// GVLs/HgGVL_Errors
// Contains common shared errors used in the mercury framework.
{attribute 'qualified_only'}
VAR_GLOBAL CONSTANT
	NO_ERROR 					: HgT_Error := HgF_CreateError(FALSE,HgE_ErrorCodes.ERR_NO_ERROR, 'No Error.', 0);
	TYPE_MISMATCH 				: HgT_Error := HgF_CreateError(TRUE, HgE_ErrorCodes.ERR_TYPE_MISMATCH, 'Type mismatch.', 0);
	SIZE_MISMATCH				: HgT_Error := HgF_CreateError(TRUE, HgE_ErrorCodes.ERR_SIZE_MISMATCH, 'Size mismatch.', 0);
	OUT_OF_BOUNDS				: HgT_Error := HgF_CreateError(TRUE, HgE_ErrorCodes.ERR_OUT_OF_BOUNDS, 'Value is outside the valid range.', 0);
	INVALID_INTERFACE  			: HgT_Error := HgF_CreateError(TRUE, HgE_ErrorCodes.ERR_INVALID_INTERFACE, 'Invalid or unknown interface.', 0);
	INVALID_REFERENCE  			: HgT_Error := HgF_CreateError(TRUE, HgE_ErrorCodes.ERR_INVALID_REFERENCE, 'Dereferencing an IEC reference in IecVarAccess failed due to an invalid destination address, e.g., NULL.', 0);
	INVALID_POINTER  			: HgT_Error := HgF_CreateError(TRUE, HgE_ErrorCodes.ERR_INVALID_POINTER, 'Invalid pointer.', 0);
	INVALID_CONVERSION  		: HgT_Error := HgF_CreateError(TRUE, HgE_ErrorCodes.ERR_INVALID_CONVERSION, 'Invalid data conversion.', 0);
	INVALID_COMPARISON  		: HgT_Error := HgF_CreateError(TRUE, HgE_ErrorCodes.ERR_INVALID_COMPARISON, 'Invalid comparison.', 0);
	INVALID_INPUT 				: HgT_Error := HgF_CreateError(TRUE, HgE_ErrorCodes.ERR_INVALID_INPUT, 'Invalid or unexpected input provided.', 0);
	MEMORY_ALLOCATION_FAILED 	: HgT_Error := HgF_CreateError(TRUE, HgE_ErrorCodes.ERR_MEMORY_ALLOCATION_FAILED, 'Memory allocation failed.', 0);
	INSUFFICIENT_MEMORY			: HgT_Error := HgF_CreateError(TRUE, HgE_ErrorCodes.ERR_INSUFFICIENT_MEMORY, 'Insufficient memory to carry out the request.', 0);
	OPERATION_FAILED			: HgT_Error := HgF_CreateError(TRUE, HgE_ErrorCodes.ERR_OPERATION_FAILED, 'Operation failed.', 0);
	INVALID_OPERATION			: HgT_Error := HgF_CreateError(TRUE, HgE_ErrorCodes.ERR_INVALID_OPERATION, 'Invalid Operation.', 0);
END_VAR

// PARAMs/HgPARAM_Constants
{attribute 'qualified_only'}
VAR_GLOBAL CONSTANT
	STR_SIZE : HgT_Size := 80; // Size of general string.
	SSTR_SIZE : HgT_Size := 40; // Size of short string.
	LSTR_SIZE : HgT_Size := 255; // Size of long string.
	INFO_SCAN_SIZE : HgT_Size := 15_000; // How many bytes to scan when looking for information. e.g. it's used by HgFB_Object to find the size of a child object in static memory.
END_VAR

// Version/Global_Version
{attribute 'TcGenerated'}
{attribute 'no-analysis'}
{attribute 'linkalways'}
// This function has been automatically generated from the project information.
VAR_GLOBAL CONSTANT
	{attribute 'const_non_replaced'}
	stLibVersion_Hg_Core : ST_LibVersion := (iMajor := 0, iMinor := 0, iBuild := 0, iRevision := 17, nFlags := 0, sVersion := '0.0.0.17');
END_VAR

// ITFs/HgI_Cloneable
INTERFACE HgI_Cloneable EXTENDS HgI_Object

// Creates a clone of the current object in dynamic memory.
METHOD Clone : HgI_Object
VAR_OUTPUT
	e : HgT_Error;
END_VAR
END_METHOD

END_INTERFACE

// ITFs/HgI_Object
// Generic interface that defines the basic properties and methods of an object in the mercury framework.
INTERFACE HgI_Object EXTENDS HgI_Queryable

// Pointer to the object in memory.
PROPERTY Address : HgT_Ptr
GET
END_GET
END_PROPERTY

// Gets the instance name of the object.
// NOTE: This only works of the object is in static memory.
METHOD GetInstanceName : HgT_LStr
VAR_OUTPUT
	e : HgT_Error;
END_VAR
END_METHOD

// Gets the instance path of the object.
// NOTE: This only works of the object is in static memory.
METHOD GetInstancePath : HgT_LStr
VAR_OUTPUT
	e : HgT_Error;
END_VAR
END_METHOD

// Returns a string representation of the object.
METHOD GetString : HgT_LStr
VAR_OUTPUT
	e : HgT_Error;
END_VAR
END_METHOD

// Gets the type name of the object as a string.
METHOD GetTypeName : HgT_Str
VAR_OUTPUT
	e : HgT_Error;
END_VAR
END_METHOD

// Checks if the current object is the same as (reference-wise) object as the input object.
METHOD Is : BOOL
VAR_INPUT
	ipObject : HgI_Object;
END_VAR
END_METHOD

// Memory area that the object is allocated in.
PROPERTY MemoryArea : HgT_MemArea
GET
END_GET
END_PROPERTY

//  Size of the object in bytes.
PROPERTY Size : HgT_Size
GET
END_GET
END_PROPERTY

END_INTERFACE

// ITFs/HgI_Queryable
// Root interface of all objects in the mercury framework. 
// Inherits __SYSTEM.IQueryInterface which is used to query an object interface/pointer for one of its interfaces.
INTERFACE HgI_Queryable EXTENDS __SYSTEM.IQueryInterface

END_INTERFACE

// ITFs/HgI_Configurable
// Base interface for a configurable system.
INTERFACE HgI_Configurable EXTENDS HgI_Object

END_INTERFACE

// ITFs/HgI_Configurator
// Base interface for a system configurator.
INTERFACE HgI_Configurator EXTENDS HgI_Object

END_INTERFACE

// ITFs/HgI_Controller
// Base interface for a controller.
INTERFACE HgI_Controller EXTENDS HgI_Object

END_INTERFACE

// ITFs/HgI_CopyableFrom
INTERFACE HgI_CopyableFrom EXTENDS HgI_Object

// Copies data to the current object from another object. Returns reference to self for method chaining.
METHOD CopyFrom : HgI_CopyableFrom
VAR_INPUT
	ipObject : HgI_Object; // Object to copy data from.
END_VAR
VAR_OUTPUT
	e : HgT_Error;
END_VAR
END_METHOD

END_INTERFACE

// ITFs/HgI_CopyableTo
INTERFACE HgI_CopyableTo EXTENDS HgI_Object

// Copies data from the current object to another object. Returns reference to self for method chaining.
METHOD CopyTo : HgI_CopyableTo
VAR_INPUT
	ipObject : HgI_Object; // Object to copy data to.
END_VAR
VAR_OUTPUT
	e : HgT_Error;
END_VAR
END_METHOD

END_INTERFACE

// ITFs/HgI_Error
// General interface for error classes in the mercury framework.
INTERFACE HgI_Error EXTENDS HgI_Queryable

// Error code specific to the particular error.
PROPERTY Code : HgT_ErrCode
GET
END_GET
END_PROPERTY

// Textual information describing the error.
PROPERTY Source : HgT_LStr
GET
END_GET
END_PROPERTY

// Indicates if an error has occurred | TRUE = error, FALSE = no error.
PROPERTY Status : BOOL
GET
END_GET
END_PROPERTY

END_INTERFACE

// ITFs/HgI_ErrorBuilder
// Interface for an error builder.
INTERFACE HgI_ErrorBuilder EXTENDS HgI_Object

// Appends the instance path of the caller to the source in the format <Caller::{caller instance path}>.
// NOTE: If the caller's interface is invalid; i.e. ipObject = 0, it will be ignored. 
METHOD AppendCallerToSource : HgI_ErrorBuilder
VAR_INPUT
	ipCaller : HgI_Object;
END_VAR
END_METHOD

// Appends a string to the error source.
METHOD AppendToSource : HgI_ErrorBuilder
VAR_INPUT
	Value : HgT_LStr;
END_VAR
END_METHOD

// Error code specific to the particular error.
PROPERTY Code : HgT_ErrCode
GET
END_GET
SET
END_SET
END_PROPERTY

// Returns the built error.
METHOD GetError : HgFB_Error
VAR_INPUT
END_VAR
END_METHOD

// Prepends a string to the error source.
METHOD PrependToSource : HgI_ErrorBuilder
VAR_INPUT
	Value : HgT_LStr;
END_VAR
END_METHOD

// Resets the built error.
METHOD Reset : HgI_ErrorBuilder
VAR_INPUT
END_VAR
END_METHOD

// Sets the error code of the error.
METHOD SetCode : HgI_ErrorBuilder
VAR_INPUT
	Code : HgT_ErrCode;
END_VAR
END_METHOD

// Sets the error in the error builder.
METHOD SetError : HgI_ErrorBuilder
VAR_INPUT
	Error : HgT_Error;
END_VAR
END_METHOD

// Sets the error source of the error.
METHOD SetSource : HgI_ErrorBuilder
VAR_INPUT
	Source : HgT_LStr;
END_VAR
END_METHOD

// Sets the status of the error
METHOD SetStatus : HgI_ErrorBuilder
VAR_INPUT
	bStatus : BOOL;
END_VAR
END_METHOD

// Textual information describing the error.
PROPERTY Source : HgT_LStr
GET
END_GET
SET
END_SET
END_PROPERTY

// Indicates if an error has occurred | TRUE = error, FALSE = no error.
PROPERTY Status : BOOL
GET
END_GET
SET
END_SET
END_PROPERTY

END_INTERFACE

// POUs/Function Blocks/HgFB_Error
// HgFB_Error is the base function block used for error handling and reporting within the mercury framework.
{attribute 'enable_dynamic_creation'}
{attribute 'no_explicit_call' := 'direct call for this function block is not allowed'}
FUNCTION_BLOCK HgFB_Error IMPLEMENTS HgI_Error
VAR
	_Status : BOOL;
	_Code : HgT_ErrCode;
	_Source : HgT_LStr;
END_VAR

// Error code specific to the particular error.
PROPERTY Code : HgT_ErrCode
GET
Code := THIS^._Code;
END_GET
END_PROPERTY

// Textual information describing the error.
PROPERTY Source : HgT_LStr
GET
Source := THIS^._Source;
END_GET
END_PROPERTY

// Indicates if an error has occurred | TRUE = error, FALSE = no error.
PROPERTY Status : BOOL
GET
Status := THIS^._Status;
END_GET
END_PROPERTY

END_FUNCTION_BLOCK

// ITFs/HgI_Status
// Base interface for a system status information.
INTERFACE HgI_Status EXTENDS HgI_Object

END_INTERFACE

// ITFs/HgI_StatusProvider
// Base interface for a system that can provide status.
INTERFACE HgI_StatusProvider EXTENDS HgI_Object

END_INTERFACE

// POUs/Function Blocks/HgFB_CycleChanged
// Function block that can be used to indicate if a the current task cycle it is instantated at has changed.
{attribute 'enable_dynamic_creation'}
{attribute 'reflection'}
{attribute 'no_explicit_call' := 'direct call for this function block is not allowed'} 
FUNCTION_BLOCK FINAL HgFB_CycleChanged EXTENDS HgFB_Object
VAR
	_nCycleLastCalled : UDINT := 4294967295; // The last cycle checked for change-in-plc-cycle.
	_nTaskIndex : DINT := HgF_GetPlcTaskInformation().TaskIndex; // The task index the function block was instantiated on.
END_VAR

// A string that represents the type of the object if the object is created dynamically.
// Function blocks intended for dynamic use must override this property.
PROPERTY PROTECTED DynamicTypeName : HgT_Str
GET
DynamicTypeName := 'HgFB_CycleChanged';
END_GET
END_PROPERTY

// Flag to indicate if cycle the cycle the function block was instantiated at has changed | TRUE = Cycle has changed.
PROPERTY _ : BOOL
GET
VAR
	nTmp : UDINT;
END_VAR
nTmp := THIS^.GetCurrentCycle();

_ := THIS^.CycleLastChecked <> nTmp;

THIS^._nCycleLastCalled := nTmp;
END_GET
END_PROPERTY

// The last cycle checked for change-in-plc-cycle.
PROPERTY CycleLastChecked : UDINT
GET
CycleLastChecked := THIS^._nCycleLastCalled;
END_GET
END_PROPERTY

// Indicates whether this is the first cycle of the task the function block was instatiated at | TRUE = first cycle.
PROPERTY FirstCycle : BOOL
GET
 FirstCycle := TwinCAT_SystemInfoVarList._TaskInfo[THIS^._nTaskIndex].FirstCycle;
END_GET
END_PROPERTY

// The current cycle of the task the function block was instatiated on.
METHOD GetCurrentCycle : UDINT
VAR_INPUT
END_VAR
GetCurrentCycle := TwinCAT_SystemInfoVarList._TaskInfo[THIS^._nTaskIndex].CycleCount;
END_METHOD

// Returns a string representation of the object.
METHOD GetString : HgT_LStr
VAR_OUTPUT
	e : HgT_Error;
END_VAR
GetString := TO_STRING(THIS^._);
END_METHOD

// Size of the object in bytes.
PROPERTY Size : HgT_Size
GET
Size := SIZEOF(THIS^);
END_GET
END_PROPERTY

// The task index the function block is instatiated on.
PROPERTY TaskIndex : DINT
GET
TaskIndex := THIS^._nTaskIndex;
END_GET
END_PROPERTY

END_FUNCTION_BLOCK

// POUs/Function Blocks/HgFB_Object
// Base function block of all mercury function blocks in the mercury framework.
{attribute 'enable_dynamic_creation'}
{attribute 'reflection'}
{attribute 'no_assign'}
{attribute 'no_explicit_call' := 'direct call for this function block is not allowed'} 
FUNCTION_BLOCK HgFB_Object IMPLEMENTS HgI_Object
VAR
END_VAR

// A string that represents the type of the object if the object is created dynamically.
// Function blocks intended for dynamic use must override this property.
PROPERTY PROTECTED DynamicTypeName : HgT_Str
GET
DynamicTypeName := 'HgFB_Object';
END_GET
END_PROPERTY

// Private local variable that acts as a flag to indicate that the size of the object may need to be recomputed.
PROPERTY PRIVATE RecomputeSize : REFERENCE TO BOOL
GET
VAR_INST
	bRecomputeSize : BOOL;
END_VAR
RecomputeSize REF= bRecomputeSize;
END_GET
END_PROPERTY

// Pointer to the object in memory.
PROPERTY FINAL Address : HgT_Ptr
GET
Address := THIS;
END_GET
END_PROPERTY

{attribute 'hide'}
METHOD FB_init : BOOL
VAR_INPUT
	bInitRetains : BOOL; // if TRUE, the retain variables are initialized (warm start / cold start)
	bInCopyCode : BOOL;  // if TRUE, the instance afterwards gets moved into the copy code (online change)
END_VAR
// Raise the recompute size flag whenever an online change is made.
// Please don't remove the 'IF' block because you think it should be 'THIS^.RecomputeSize := bInCopyCode;'
// This is done on purpose to latch the flag. Only the size property should reset it.
IF bInCopyCode THEN THIS^.RecomputeSize := bInCopyCode; END_IF
END_METHOD

{attribute 'hide'}
METHOD FB_reinit : BOOL
VAR_INPUT
END_VAR
END_METHOD

// Gets the instance name of the object.
// NOTE: This only works of the object is in static memory.
METHOD FINAL GetInstanceName : HgT_LStr
VAR_OUTPUT
	e : HgT_Error;
END_VAR
CASE THIS^.MemoryArea OF
	HgT_MemArea.Static: 
		GetInstanceName := HgF_GetVariableNameByAddress(THIS, THIS^.Size, e => e);
	HgT_MemArea.Dynamic:
		GetInstanceName := '<Dynamic>';
	HgT_MemArea.CNC:
		GetInstanceName := '<Unsupported>';
ELSE
	GetInstanceName := '<Unknown>';
	e := HgF_CreateError(TRUE, HgE_ErrorCodes.ERR_OPERATION_FAILED, 'Cannot identify the memory area of the object.', 0);
	END_CASE
END_METHOD

// Gets the instance path of an object.
// NOTE: This only works of the object is in static memory.
METHOD FINAL GetInstancePath : HgT_LStr
VAR_OUTPUT
	e : HgT_Error;
END_VAR
CASE THIS^.MemoryArea OF
	HgT_MemArea.Static: 
		GetInstancePath := HgF_GetVariablePathByAddress(THIS, THIS^.Size, e => e);
	HgT_MemArea.Dynamic:
		GetInstancePath := '<Dynamic>';
	HgT_MemArea.CNC:
		GetInstancePath := '<Unsupported>';
ELSE
	GetInstancePath := '<Unknown>';
	e := HgF_CreateError(TRUE, HgE_ErrorCodes.ERR_OPERATION_FAILED, 'Cannot identify the memory area of the object.', 0);
	END_CASE
END_METHOD

// Returns a string representation of the object.
{attribute 'TcRpcEnable'}
METHOD GetString : HgT_LStr
VAR_OUTPUT
	e : HgT_Error;
END_VAR
GetString := THIS^.GetTypeName(e => e);

IF e.Status THEN RETURN; END_IF

GetString := Tc2_Standard.CONCAT(GetString, CONCAT(' at ', TO_STRING(THIS)));
END_METHOD

// Gets the type name of the object as a string.
METHOD FINAL GetTypeName : HgT_Str
VAR_OUTPUT
	e : HgT_Error;
END_VAR
CASE THIS^.MemoryArea OF
	HgT_MemArea.Static: 
		GetTypeName := HgF_GetTypeNameByAddress(THIS, THIS^.Size, e => e);
	HgT_MemArea.Dynamic:
		GetTypeName := THIS^.DynamicTypeName;
	HgT_MemArea.CNC:
		GetTypeName := '<Unsupported>';
ELSE
	GetTypeName := '<Unknown>';
	END_CASE
END_METHOD

// Checks if the current object is the same as (reference-wise) object as the input object.
METHOD FINAL Is : BOOL
VAR_INPUT
	ipObject : HgI_Object;
END_VAR
Is := SEL(ipObject <> 0, FALSE, ipObject.Address = THIS);
END_METHOD

// Memory area that the object is allocated in.
PROPERTY FINAL MemoryArea : HgT_MemArea
GET
MemoryArea := Tc2_System.F_CheckMemoryArea(THIS, 1);
END_GET
END_PROPERTY

// Size of the object in bytes.
PROPERTY Size : HgT_Size
GET
VAR_INST
	_Size : HgT_Size;
END_VAR
IF _Size > 0 AND NOT(THIS^.RecomputeSize) THEN Size := _Size; RETURN; END_IF

// Set the recompute flag to false.
THIS^.RecomputeSize := FALSE;

CASE THIS^.MemoryArea OF
// Attempt to get size of object.
	HgT_MemArea.Static:
	// If object is in static memory try and look for it using the TcCOM object server and get it's size.
		FOR _Size := SIZEOF(THIS^) TO HgPARAM_Constants.INFO_SCAN_SIZE DO
			IF HgF_GetTypeNameByAddress(THIS, _Size) <> '' THEN RETURN; END_IF
			END_FOR
	END_CASE
	
// In any other case just return the base object size.
_Size := SIZEOF(THIS^);
END_GET
END_PROPERTY

END_FUNCTION_BLOCK

// POUs/Functions/HgF_GetVariableNameByAddress
// Returns the name of a variable as a string using its pointer and size.
// Variables allocated in dynamic memory are not supported.
FUNCTION HgF_GetVariableNameByAddress : HgT_LStr
VAR_INPUT
	Address : HgT_Ptr; // Pointer to variable.
	Size : HgT_Size; // Size of variable in bytes.
END_VAR
VAR_OUTPUT
	e : HgT_Error;
END_VAR
VAR
	_pCursor : POINTER TO BYTE;
	_pVariableName : POINTER TO HgT_LStr;
END_VAR

HgF_GetVariableNameByAddress := HgF_GetVariablePathByAddress(Address, Size, e => e);

IF e.Status OR_ELSE HgF_GetVariableNameByAddress = '' THEN RETURN; END_IF

_pCursor := ADR(HgF_GetVariableNameByAddress);

REPEAT
	IF _pCursor^ = 46 THEN _pVariableName := _pCursor + 1; END_IF
	_pCursor := _pCursor + 1;
UNTIL
	_pCursor^ = 0
	END_REPEAT

HgF_GetVariableNameByAddress := SEL(_pVariableName = 0, _pVariableName^, HgF_GetVariableNameByAddress);

END_FUNCTION

// POUs/Functions/HgF_GetVariablePathByAddress
// Returns the path of a variable as a string using its pointer and size.
// Variables allocated in dynamic memory are not supported.
{warning disable C0394}
FUNCTION HgF_GetVariablePathByAddress : HgT_LStr
VAR_INPUT
	Address : HgT_Ptr; // Pointer to variable.
	Size : HgT_Size; // Size of variable in bytes.
END_VAR
VAR_OUTPUT
	e : HgT_Error;
END_VAR
VAR
	_nTmp : UDINT := SIZEOF(HgF_GetVariablePathByAddress);
	_ipComInterface : ITcIecApplicationInfo := HgF_TcComIecApplicationInfo().GetInterface(e => e);;
	_Result : HRESULT;
END_VAR

IF _ipComInterface <> 0 THEN
	_Result := _ipComInterface.GetSymbolNameByAddress(TO_UDINT(Size), Address, _nTmp, ADR(HgF_GetVariablePathByAddress));
	e := SEL(
		Tc3_Module.SUCCEEDED(_Result),
		HgF_CreateError(TRUE, _Result, 'Failed to get variable path. Check error code against "Tc3_Module/Error Codes" section on infosys.', 0),
		HgGVL_Errors.NO_ERROR);
	END_IF

END_FUNCTION

// POUs/Functions/HgF_CreateError
// Function for creating an error function block.
// If ipObject object is not 0 the instance path will be appended to the error message.
FUNCTION HgF_CreateError : HgFB_Error
VAR_INPUT
	bStatus : BOOL; // Indicates if an error has occurred | TRUE = error, FALSE = no error.
	Code : HgT_ErrCode; // Error code specific to the particular error.
	Source : HgT_LStr; // Textual information describing the error.
	ipCaller : HgI_Object; // Object that created the error, set to 0 if you don't want append caller to error message.
END_VAR
VAR
	_fbError : HgFB_MutableError;
END_VAR

_fbError.Status := bStatus;
_fbError.Code := Code;
_fbError.Source := Source;

HgF_CreateError := _fbError.AppendCaller(ipCaller);

END_FUNCTION

// POUs/Function Blocks/HgFB_MutableError
// Base function block for mutable errors used for error handling and reporting within the mercury framework.
{attribute 'enable_dynamic_creation'}
{attribute 'no_explicit_call' := 'direct call for this function block is not allowed'}
FUNCTION_BLOCK HgFB_MutableError EXTENDS HgFB_Error IMPLEMENTS HgI_Error
VAR
END_VAR

METHOD FINAL AppendCaller : REFERENCE TO HgFB_MutableError
VAR_INPUT
	ipCaller : HgI_Object;
END_VAR
AppendCaller REF= THIS^;
IF ipCaller = 0 THEN RETURN; END_IF

THIS^._Source := CONCAT(THIS^._Source, CONCAT(' <Caller::', CONCAT(ipCaller.GetInstancePath(),'>')));
END_METHOD

// Error code specific to the particular error.
PROPERTY FINAL Code : HgT_ErrCode
SET
THIS^._Code := Code;
END_SET
END_PROPERTY

// Textual information describing the error.
PROPERTY FINAL Source : HgT_LStr
SET
THIS^._Source := Source;
END_SET
END_PROPERTY

// Indicates if an error has occurred | TRUE = error, FALSE = no error.
PROPERTY FINAL Status : BOOL
SET
THIS^._Status := Status;
END_SET
END_PROPERTY

END_FUNCTION_BLOCK

// POUs/Functions/HgF_TcComIecApplicationInfo
// Function that acts as a singleton for HgFB_TcComIecApplicationInfo, a function block that that manages the ITcIecApplicationInfo TcCOM Interface used by Hg_Core.
FUNCTION HgF_TcComIecApplicationInfo : REFERENCE TO HgFB_TcComIecApplicationInfo
VAR_STAT
	_fbTcComIecApplicationInfo : HgFB_TcComIecApplicationInfo;
END_VAR

HgF_TcComIecApplicationInfo REF= _fbTcComIecApplicationInfo;

END_FUNCTION

// POUs/Function Blocks/HgFB_TcComIecApplicationInfo
// Function block that manages the ITcIecApplicationInfo TcCOM Interface used by Hg_Core.
{attribute 'enable_dynamic_creation'}
{attribute 'no_assign'}
{attribute 'no_explicit_call' := 'direct call for this function block is not allowed'} 
FUNCTION_BLOCK FINAL HgFB_TcComIecApplicationInfo IMPLEMENTS HgI_Queryable
VAR
	_ipIecApplicationInformation : ITcIecApplicationInfo;
	_hIecApplicationInformation : HRESULT := Tc3_Module.GVL.E_FAIL;
END_VAR

{attribute 'hide'}
METHOD FB_exit : BOOL
VAR_INPUT
	bInCopyCode : BOOL; // if TRUE, the exit method is called for exiting an instance that is copied afterwards (online change).
END_VAR
// no online change
IF bInCopyCode THEN RETURN; END_IF

// Safe release of ITcIecApplicationInfo.
Tc3_Module.FW_SafeRelease(ADR(THIS^._ipIecApplicationInformation));
THIS^._hIecApplicationInformation := Tc3_Module.GVL.E_FAIL;
END_METHOD

{attribute 'hide'}
{attribute 'no_explicit_call' := 'direct call for this method is not allowed'}
METHOD FB_init : BOOL
VAR_INPUT
	bInitRetains : BOOL; // if TRUE, the retain variables are initialized (warm start / cold start)
	bInCopyCode : BOOL;  // if TRUE, the instance afterwards gets moved into the copy code (online change)
END_VAR
// No online change.
IF bInCopyCode THEN RETURN; END_IF

// Get instance of ITcIecApplicationInfo.
THIS^._hIecApplicationInformation := Tc3_Module.FW_ObjMgr_GetObjectInstance(
	TwinCAT_SystemInfoVarList._AppInfo.ObjId, 
	TC_GLOBAL_IID_LIST.IID_ITcIecApplicationInfo, 
	ADR(THIS^._ipIecApplicationInformation)
);
END_METHOD

METHOD GetInterface : ITcIecApplicationInfo
VAR_OUTPUT
	e : HgT_Error;
END_VAR
// If instance of ITcIecApplicationInfo failed to be obtained on 
// FB_init or FB_exit was explicitly called try to get it gain.


IF Tc3_Module.FAILED(THIS^._hIecApplicationInformation) THEN
	THIS^._hIecApplicationInformation := Tc3_Module.FW_ObjMgr_GetObjectInstance(
		TwinCAT_SystemInfoVarList._AppInfo.ObjId, 
		TC_GLOBAL_IID_LIST.IID_ITcIecApplicationInfo, 
		ADR(THIS^._ipIecApplicationInformation)
	);
	END_IF

e := SEL(
	Tc3_Module.SUCCEEDED(THIS^._hIecApplicationInformation),
	HgF_CreateError(TRUE, THIS^._hIecApplicationInformation, 'No failed to get interface. Check error code against "Tc3_Module/Error Codes" section on infosys.', 0),
	HgGVL_Errors.NO_ERROR);

GetInterface := THIS^._ipIecApplicationInformation;
END_METHOD

END_FUNCTION_BLOCK

// POUs/Functions/HgF_GetTypeNameByAddress
// Returns the datatype of a variable as a string using its pointer and size.
// Variables allocated in dynamic memory are not supported.
FUNCTION HgF_GetTypeNameByAddress : HgT_Str
VAR_INPUT
	Address :HgT_Ptr; // Pointer to variable.
	Size : HgT_Size; // Size of variable in bytes.
END_VAR
VAR_OUTPUT
	e : HgT_Error;
END_VAR
VAR 
	_nTmp : UDINT := SIZEOF(HgF_GetTypeNameByAddress);
	_ipComInterface : ITcIecApplicationInfo := HgF_TcComIecApplicationInfo().GetInterface(e => e);;
	_Result : HRESULT;
END_VAR


	
IF _ipComInterface <> 0 THEN
	_Result := _ipComInterface.GetDatatypeNameByAddress(TO_UDINT(Size), Address, _nTmp, ADR(HgF_GetTypeNameByAddress));
	e := SEL(
		Tc3_Module.SUCCEEDED(_Result),
		HgF_CreateError(TRUE, _Result, 'Failed to get variable typename. Check error code against "Tc3_Module/Error Codes" section on infosys.', 0),
		HgGVL_Errors.NO_ERROR);
	END_IF

END_FUNCTION

// POUs/Functions/HgF_GetPlcTaskInformation
// Retrieves the current plc task's information.
FUNCTION HgF_GetPlcTaskInformation : REFERENCE TO HgT_PlcTaskInfo
VAR
	_fbGetCurrentTaskIndex : GETCURTASKINDEX;
	_PlcTaskSysInfo : PlcTaskSystemInfo;
END_VAR
VAR_STAT
	_PlcTaskInformation : HgT_PlcTaskInfo;
END_VAR

_fbGetCurrentTaskIndex();
_PlcTaskSysInfo := TwinCAT_SystemInfoVarList._TaskInfo[_fbGetCurrentTaskIndex.index];
_PlcTaskInformation.AdsPort 				:= _PlcTaskSysInfo.AdsPort;
_PlcTaskInformation.CycleCount 				:= _PlcTaskSysInfo.CycleCount;
_PlcTaskInformation.CycleTime 				:= TO_LTIME(_PlcTaskSysInfo.CycleTime*100);
_PlcTaskInformation.CycleTimeExceeded 		:= _PlcTaskSysInfo.CycleTimeExceeded;
_PlcTaskInformation.DcTaskTime 				:= _PlcTaskSysInfo.DcTaskTime;
_PlcTaskInformation.FirstCycle				:= _PlcTaskSysInfo.FirstCycle;
_PlcTaskInformation.InCallAfterOutputUpdate := _PlcTaskSysInfo.InCallAfterOutputUpdate;
_PlcTaskInformation.LastExecTime 			:= TO_LTIME(_PlcTaskSysInfo.LastExecTime*100);
_PlcTaskInformation.ObjId 					:= _PlcTaskSysInfo.ObjId;
_PlcTaskInformation.Priority 				:= _PlcTaskSysInfo.Priority;
_PlcTaskInformation.RTViolation 			:= _PlcTaskSysInfo.RTViolation;
_PlcTaskInformation.TaskName 				:= _PlcTaskSysInfo.TaskName;
_PlcTaskInformation.TaskIndex 				:= _fbGetCurrentTaskIndex.Index;

HgF_GetPlcTaskInformation REF= _PlcTaskInformation;

END_FUNCTION

// POUs/Function Blocks/HgFB_ErrorBuilder
// Function block for building an error.
{attribute 'enable_dynamic_creation'}
{attribute 'no_explicit_call' := 'direct call for this function block is not allowed'} 
FUNCTION_BLOCK FINAL HgFB_ErrorBuilder EXTENDS HgFB_Object IMPLEMENTS HgI_ErrorBuilder
VAR
	// Working error.
	_Error : HgFB_MutableError;
END_VAR

// Appends the instance path of the caller to the source in the format <Caller::{caller instance path}>.
// NOTE: If the caller's interface is invalid; i.e. ipObject = 0, it will be ignored. 
METHOD AppendCallerToSource : HgI_ErrorBuilder
VAR_INPUT
	ipCaller : HgI_Object;
END_VAR
AppendCallerToSource := THIS^;

THIS^._Error.AppendCaller(ipCaller);
END_METHOD

// Appends a string to the error source.
METHOD AppendToSource : HgI_ErrorBuilder
VAR_INPUT
	Value : HgT_LStr;
END_VAR
AppendToSource := THIS^;

THIS^._Error.Source := Tc2_Standard.CONCAT(THIS^._Error.Source, Value);
END_METHOD

// Error code specific to the particular error.
PROPERTY Code : HgT_ErrCode
GET
Code := THIS^._Error.Code;
END_GET
SET
THIS^._Error.Code := Code;
END_SET
END_PROPERTY

// A string that represents the type of the object if the object is created dynamically.
// Function blocks intended for dynamic use must override this property.
PROPERTY PROTECTED DynamicTypeName : HgT_Str
GET
DynamicTypeName := 'HgFB_ErrorBuilder';
END_GET
END_PROPERTY

// Returns the built error.
{attribute 'TcRpcEnable'}
METHOD GetError : HgFB_Error
VAR_INPUT
END_VAR
GetError := THIS^._Error;
END_METHOD

// Returns a string representation of the object.
{attribute 'TcRpcEnable'}
{warning disable C0394}
METHOD GetString : HgT_LStr
VAR_OUTPUT
	e : HgT_Error;
END_VAR
VAR
	fbJson : Tc3_JsonXml.FB_JsonSaxWriter;
	Result : HRESULT;
END_VAR
fbJson.StartObject();
fbJson.AddKey('Status');
fbJson.AddBool(THIS^._Error.Status);
fbJson.AddKey('Code');
fbJson.AddLint(THIS^._Error.Code);
fbJson.AddKey('Source');
GetString := THIS^._Error.Source;
fbJson.AddString(GetString);
fbJson.EndObject();
GetString := fbJson.GetDocument(hrErrorCode => Result);
e := SEL(
	Tc3_Module.SUCCEEDED(Result),
	HgF_CreateError(TRUE, Result, 'Failed to generate json. Check error code against "Tc3_Module/Error Codes" section on infosys.', 0),
	HgGVL_Errors.NO_ERROR);
END_METHOD

// Prepends a string to the error source.
METHOD PrependToSource : HgI_ErrorBuilder
VAR_INPUT
	Value : HgT_LStr;
END_VAR
PrependToSource := THIS^;

THIS^._Error.Source := Tc2_Standard.CONCAT(Value, THIS^._Error.Source);
END_METHOD

// Resets the built error.
METHOD Reset : HgI_ErrorBuilder
VAR_INPUT
END_VAR
Reset := THIS^;

THIS^._Error.Status := FALSE;
THIS^._Error.Code := 0;
THIS^._Error.Source := '';
END_METHOD

// Sets the error code of the error.
METHOD SetCode : HgI_ErrorBuilder
VAR_INPUT
	Code : HgT_ErrCode;
END_VAR
SetCode := THIS^;

THIS^._Error.Code := Code;
END_METHOD

// Sets the error in the error builder.
METHOD SetError : HgI_ErrorBuilder
VAR_INPUT
	Error : HgT_Error;
END_VAR
SetError := THIS^;

THIS^._Error.Status := Error.Status;
THIS^._Error.Code := Error.Code;
THIS^._Error.Source := Error.Source;
END_METHOD

// Sets the error source of the error.
METHOD SetSource : HgI_ErrorBuilder
VAR_INPUT
	Source : HgT_LStr;
END_VAR
SetSource := THIS^;

THIS^._Error.Source := Source;
END_METHOD

// Sets the status of the error
METHOD SetStatus : HgI_ErrorBuilder
VAR_INPUT
	bStatus : BOOL;
END_VAR
SetStatus := THIS^;

THIS^._Error.Status := bStatus;
END_METHOD

PROPERTY Size : HgT_Size
GET
Size := SIZEOF(THIS^);
END_GET
END_PROPERTY

// Textual information describing the error.
PROPERTY Source : HgT_LStr
GET
Source := THIS^._Error.Source;
END_GET
SET
THIS^._Error.Source := Source;
END_SET
END_PROPERTY

// Indicates if an error has occurred | TRUE = error, FALSE = no error.
PROPERTY Status : BOOL
GET
Status := THIS^._Error.Status;
END_GET
SET
THIS^._Error.Status := Status;
END_SET
END_PROPERTY

END_FUNCTION_BLOCK

// POUs/Function Blocks/HgFB_FirstCall
// Function block that can be used to indicate whether a section of code has been running for the first time.
{attribute 'enable_dynamic_creation'}
{attribute 'reflection'}
{attribute 'no_explicit_call' := 'direct call for this function block is not allowed'} 
FUNCTION_BLOCK FINAL HgFB_FirstCall EXTENDS HgFB_Object
VAR
	_CallFlag : BOOL := TRUE; 
END_VAR

// Flag to indicate if code section is running for the first time | TRUE = Called for the first time.
PROPERTY _ : BOOL
GET
_ := THIS^._CallFlag;

THIS^._CallFlag := FALSE;
END_GET
END_PROPERTY

// A string that represents the type of the object if the object is created dynamically.
// Function blocks intended for dynamic use must override this property.
PROPERTY PROTECTED DynamicTypeName : HgT_Str
GET
DynamicTypeName := 'HgFB_FirstCall';
END_GET
END_PROPERTY

// Returns a string representation of the object.
METHOD GetString : HgT_LStr
VAR_OUTPUT
	e : HgT_Error;
END_VAR
GetString := TO_STRING(THIS^._);
END_METHOD

// Resets the flag for first call.
METHOD Reset
VAR_INPUT
END_VAR
THIS^._CallFlag := TRUE;
END_METHOD

PROPERTY Size : HgT_Size
GET
Size := SIZEOF(THIS^);
END_GET
END_PROPERTY

END_FUNCTION_BLOCK

// POUs/Function Blocks/HgFB_FlagHasChanged
// Checks if the watched value has changed.
{attribute 'enable_dynamic_creation'}
{attribute 'no_explicit_call' := 'direct call for this function block is not allowed'} 
FUNCTION_BLOCK FINAL HgFB_FlagHasChanged EXTENDS HgFB_Object
VAR
	_bValue : BOOL; 
END_VAR

// A string that represents the type of the object if the object is created dynamically.
// Function blocks intended for dynamic use must override this property.
PROPERTY PROTECTED DynamicTypeName : HgT_Str
GET
DynamicTypeName := 'HgFB_FlagHasChanged';
END_GET
END_PROPERTY

// Size of the object in bytes.
PROPERTY Size : HgT_Size
GET
Size := SIZEOF(THIS^);
END_GET
END_PROPERTY

METHOD Watch : BOOL
VAR_INPUT
	Value : BOOL;
END_VAR
VAR_INST
	bFirstCall : BOOL := TRUE;
END_VAR
IF bFirstCall THEN bFirstCall := FALSE; Watch := TRUE; THIS^._bValue := Value; RETURN; END_IF

Watch := THIS^._bValue <> Value;
END_METHOD

END_FUNCTION_BLOCK

// POUs/Function Blocks/HgFB_FloatHasChanged
// Checks if the watched value has changed.
{attribute 'enable_dynamic_creation'}
{attribute 'no_explicit_call' := 'direct call for this function block is not allowed'} 
FUNCTION_BLOCK FINAL HgFB_FloatHasChanged EXTENDS HgFB_Object
VAR
	_fValue : LREAL; 
END_VAR

// A string that represents the type of the object if the object is created dynamically.
// Function blocks intended for dynamic use must override this property.
PROPERTY PROTECTED DynamicTypeName : HgT_Str
GET
DynamicTypeName := 'HgFB_FloatHasChanged';
END_GET
END_PROPERTY

// Size of the object in bytes.
PROPERTY Size : HgT_Size
GET
Size := SIZEOF(THIS^);
END_GET
END_PROPERTY

METHOD Watch : BOOL
VAR_INPUT
	fValue : LREAL;
END_VAR
VAR_INST
	bFirstCall : BOOL := TRUE;
END_VAR
IF bFirstCall THEN bFirstCall := FALSE; Watch := TRUE; THIS^._fValue := fValue; RETURN; END_IF

Watch := THIS^._fValue <> fValue;
END_METHOD

END_FUNCTION_BLOCK

// POUs/Function Blocks/HgFB_HasChanged
// Checks if the watched value has changed.
{attribute 'enable_dynamic_creation'}
{attribute 'reflection'}
{attribute 'no_explicit_call' := 'direct call for this function block is not allowed'} 
FUNCTION_BLOCK FINAL HgFB_HasChanged EXTENDS HgFB_Object
VAR
	_nHash 		: DWORD;
	_nSize		: DINT 					:= -1;
	_eTypeClass : __SYSTEM.TYPE_CLASS 	:= __SYSTEM.TYPE_CLASS.TYPE_NONE;
END_VAR

// A string that represents the type of the object if the object is created dynamically.
// Function blocks intended for dynamic use must override this property.
PROPERTY PROTECTED DynamicTypeName : HgT_Str
GET
DynamicTypeName := 'HgFB_HasChanged';
END_GET
END_PROPERTY

// Size of the object in bytes.
PROPERTY Size : HgT_Size
GET
Size := SIZEOF(THIS^);
END_GET
END_PROPERTY

METHOD Watch : BOOL
VAR_INPUT
	Value : ANY;
END_VAR
VAR
	nHash : DWORD;
END_VAR
nHash := HgF_SimpleHash(Value);

IF THIS^._nHash = nHash AND_THEN THIS^._nSize = Value.diSize AND_THEN THIS^._eTypeClass = Value.TypeClass THEN RETURN; END_IF 

THIS^._nHash 		:= nHash;
THIS^._nSize 		:= Value.diSize;
THIS^._eTypeClass 	:= Value.TypeClass;

Watch := TRUE;
END_METHOD

END_FUNCTION_BLOCK

// POUs/Functions/HgF_SimpleHash
// This function calculates a hashcode of a given value using the FNV-1a 32-bit hash algorithm. Source: http://www.isthe.com/chongo/tech/comp/fnv/
FUNCTION HgF_SimpleHash : DWORD
VAR_INPUT
	Data : ANY;
END_VAR
VAR
	i, nSize, nHash : DWORD;
END_VAR
VAR_STAT CONSTANT
	nPrime : DWORD := 16#1000193; // 32-bit FNV Prime
END_VAR

nHash := 16#811C9DC5; // 32-bit offset basis
CASE Data.TypeClass OF
	__SYSTEM.TYPE_CLASS.TYPE_STRING:
		nSize := Tc2_Utilities.LEN2(Data.pValue)- 1;
	__SYSTEM.TYPE_CLASS.TYPE_WSTRING:
		nSize := Tc2_Utilities.WLEN2(Data.pValue)*2-1;
ELSE
		nSize := TO_UDINT(Data.diSize) - 1;
END_CASE
FOR i := 0 TO nSize DO nHash :=(nHash XOR Data.pValue[i])*nPrime; END_FOR
HgF_SimpleHash := nHash;

END_FUNCTION

// POUs/Function Blocks/HgFB_IntHasChanged
// Checks if the watched value has changed.
{attribute 'enable_dynamic_creation'}
{attribute 'no_explicit_call' := 'direct call for this function block is not allowed'} 
FUNCTION_BLOCK FINAL HgFB_IntHasChanged EXTENDS HgFB_Object
VAR
	_nValue : LINT; 
END_VAR

// A string that represents the type of the object if the object is created dynamically.
// Function blocks intended for dynamic use must override this property.
PROPERTY PROTECTED DynamicTypeName : HgT_Str
GET
DynamicTypeName := 'HgFB_IntHasChanged';
END_GET
END_PROPERTY

// Size of the object in bytes.
PROPERTY Size : HgT_Size
GET
Size := SIZEOF(THIS^);
END_GET
END_PROPERTY

METHOD Watch : BOOL
VAR_INPUT
	nValue : LINT;
END_VAR
VAR_INST
	bFirstCall : BOOL := TRUE;
END_VAR
IF bFirstCall THEN bFirstCall := FALSE; Watch := TRUE; THIS^._nValue := nValue; RETURN; END_IF

Watch := THIS^._nValue <> nValue;
END_METHOD

END_FUNCTION_BLOCK

// POUs/Function Blocks/HgFB_LTimeHasChanged
// Checks if the watched value has changed.
{attribute 'enable_dynamic_creation'}
{attribute 'no_explicit_call' := 'direct call for this function block is not allowed'} 
FUNCTION_BLOCK FINAL HgFB_LTimeHasChanged EXTENDS HgFB_Object
VAR
	_tValue : LTIME; 
END_VAR

// A string that represents the type of the object if the object is created dynamically.
// Function blocks intended for dynamic use must override this property.
PROPERTY PROTECTED DynamicTypeName : HgT_Str
GET
DynamicTypeName := 'HgFB_LTimeHasChanged';
END_GET
END_PROPERTY

// Size of the object in bytes.
PROPERTY Size : HgT_Size
GET
Size := SIZEOF(THIS^);
END_GET
END_PROPERTY

METHOD Watch : BOOL
VAR_INPUT
	tValue : LTIME;
END_VAR
VAR_INST
	bFirstCall : BOOL := TRUE;
END_VAR
IF bFirstCall THEN bFirstCall := FALSE; Watch := TRUE; THIS^._tValue := tValue; RETURN; END_IF

Watch := THIS^._tValue <> tValue;
END_METHOD

END_FUNCTION_BLOCK

// POUs/Function Blocks/HgFB_TimeHasChanged
// Checks if the watched value has changed.
{attribute 'enable_dynamic_creation'}
{attribute 'no_explicit_call' := 'direct call for this function block is not allowed'} 
FUNCTION_BLOCK FINAL HgFB_TimeHasChanged EXTENDS HgFB_Object
VAR
	_tValue : TIME; 
END_VAR

// A string that represents the type of the object if the object is created dynamically.
// Function blocks intended for dynamic use must override this property.
PROPERTY PROTECTED DynamicTypeName : HgT_Str
GET
DynamicTypeName := 'HgFB_TimeHasChanged';
END_GET
END_PROPERTY

// Size of the object in bytes.
PROPERTY Size : HgT_Size
GET
Size := SIZEOF(THIS^);
END_GET
END_PROPERTY

METHOD Watch : BOOL
VAR_INPUT
	tValue : TIME;
END_VAR
VAR_INST
	bFirstCall : BOOL := TRUE;
END_VAR
IF bFirstCall THEN bFirstCall := FALSE; Watch := TRUE; THIS^._tValue := tValue; RETURN; END_IF

Watch := THIS^._tValue <> tValue;
END_METHOD

END_FUNCTION_BLOCK

// POUs/Function Blocks/HgFB_UIntHasChanged
// Checks if the watched value has changed.
{attribute 'enable_dynamic_creation'}
{attribute 'no_explicit_call' := 'direct call for this function block is not allowed'} 
FUNCTION_BLOCK FINAL HgFB_UIntHasChanged EXTENDS HgFB_Object
VAR
	_nValue : ULINT; 
END_VAR

// A string that represents the type of the object if the object is created dynamically.
// Function blocks intended for dynamic use must override this property.
PROPERTY PROTECTED DynamicTypeName : HgT_Str
GET
DynamicTypeName := 'HgFB_UIntHasChanged';
END_GET
END_PROPERTY

// Size of the object in bytes.
PROPERTY Size : HgT_Size
GET
Size := SIZEOF(THIS^);
END_GET
END_PROPERTY

METHOD Watch : BOOL
VAR_INPUT
	nValue : ULINT;
END_VAR
VAR_INST
	bFirstCall : BOOL := TRUE;
END_VAR
IF bFirstCall THEN bFirstCall := FALSE; Watch := TRUE; THIS^._nValue := nValue; RETURN; END_IF

Watch := THIS^._nValue <> nValue;
END_METHOD

END_FUNCTION_BLOCK

// POUs/Functions/HgF_AppendCallerToError
// Appends caller to current error.
FUNCTION HgF_AppendCallerToError
VAR_IN_OUT
	Error : HgT_Error;
END_VAR
VAR_INPUT
	ipCaller : HgI_Object;
END_VAR
VAR
	_fbError : HgFB_MutableError;
END_VAR

_fbError.Status := Error.Status;
_fbError.Code := Error.Code;
_fbError.Source := Error.Source;

Error := _fbError.AppendCaller(ipCaller);

END_FUNCTION

// POUs/Functions/HgF_ChangeDecimalPlaces
// Takes in an input and returnd a value rounded to the specified decimal places.
FUNCTION HgF_ChangeDecimalPlaces : LREAL
VAR_INPUT
	fValue : LREAL;
	nDecimalPlaces : USINT;
END_VAR

HgF_ChangeDecimalPlaces := TO_DINT(fValue * EXPT(10, nDecimalPlaces)) / EXPT(10, nDecimalPlaces);

END_FUNCTION

// POUs/Functions/HgF_Dealloc
// Safely releases pointer. If the pointer was allocated in dynamic memory it will be deleted if it was instatic memory it will be set to zero.
// Returns TRUE if successful 
FUNCTION HgF_Dealloc : BOOL
VAR_INPUT
	refPointer : REFERENCE TO HgT_Ptr;
END_VAR
VAR_OUTPUT
	e : HgT_Error;
END_VAR

IF NOT __ISVALIDREF(refPointer) THEN e := HgGVL_Errors.INVALID_REFERENCE; RETURN; END_IF

CASE Tc2_System.F_CheckMemoryArea(refPointer, 1) OF
	HgT_MemArea.Dynamic: __DELETE(refPointer); HgF_Dealloc := TRUE;
	HgT_MemArea.Static: refPointer := 0; HgF_Dealloc := TRUE;
ELSE
	e := HgF_CreateError(TRUE, HgE_ErrorCodes.ERR_INVALID_POINTER, 'Pointer must be located in static or dynamic memory and non zero.', 0);
	END_CASE

END_FUNCTION

// POUs/Functions/HgF_ErrorBuilder
// Function that acts as a singleton for HgFB_ErrorBuilder.
FUNCTION HgF_ErrorBuilder : HgI_ErrorBuilder
VAR_STAT
	_fbBuilder : HgFB_ErrorBuilder;
END_VAR

HgF_ErrorBuilder := _fbBuilder.Reset();

END_FUNCTION

// POUs/Functions/HgF_GetAddress
// Gets the address of an object from it's interface.
FUNCTION HgF_GetAddress : HgT_Ptr
VAR_INPUT
	ipInterface : __SYSTEM.IQueryInterface;
END_VAR
VAR
	_pInterface : POINTER TO HgT_Ptr := ADR(ipInterface);
END_VAR

IF ipInterface = 0 THEN RETURN; END_IF
HgF_GetAddress := _pInterface^ - SIZEOF(ipInterface);

END_FUNCTION

// POUs/Functions/HgF_GetInf
// Gets Infinity (Inf)
FUNCTION HgF_GetInf : LREAL
VAR_STAT
	_Inf : LREAL := TO_LREAL('#Inf');
END_VAR

HgF_GetInf := _Inf;

END_FUNCTION

// POUs/Functions/HgF_GetNaN
// Gets Not-A-Number (NaN)
FUNCTION HgF_GetNaN : LREAL
VAR_STAT
	_NaN : LREAL := TO_LREAL('#NaN');
END_VAR

HgF_GetNaN := _NaN;

END_FUNCTION

// POUs/Functions/HgF_GetSize
// Gets the size of an function block in static memory via its interface.
// Interface must inherit from  __SYSTEM.IQueryInterface or HgI_Queryable.
// NOTE: This is performance intensive. Cyclic use is not recommened.
FUNCTION HgF_GetSize : HgT_Size
VAR_INPUT
	ipInterface : __SYSTEM.IQueryInterface; // The interface of the object whose size is to be retrieved.
	ScanLength : HgT_Size; // Maximum number of bytes to scan.
END_VAR
VAR_OUTPUT
	e : HgT_Error;
END_VAR
VAR
	_Address : HgT_Ptr := HgF_GetAddress(ipInterface);
END_VAR

CASE Tc2_System.F_CheckMemoryArea(_Address, 1) OF
	HgT_MemArea.Static:
		FOR HgF_GetSize := SIZEOF(ipInterface) TO ScanLength DO
			IF HgF_GetTypeNameByAddress(_Address, HgF_GetSize) <> '' THEN RETURN; END_IF
			END_FOR
		HgF_GetTypeNameByAddress(_Address, HgF_GetSize, e => e);
		e := HgF_CreateError(TRUE, e.Code, 'Failed to get size. Check error code against "Tc3_Module/Error Codes" section on infosys.', 0);
		HgF_GetSize := 0;
		RETURN;
	END_CASE

e := HgF_CreateError(TRUE, HgE_ErrorCodes.ERR_INVALID_INPUT, 'Invalid input. Object must be in static memory and its interface must be valid.', 0);

END_FUNCTION

// POUs/Functions/HgF_GetTypeName
// Returns the datatype of a variable as a string.
// Variables allocated in dynamic memory are not supported.
FUNCTION HgF_GetTypeName : HgT_Str
VAR_INPUT
	Variable : ANY;
END_VAR
VAR_OUTPUT
	e : HgT_Error;
END_VAR

HgF_GetTypeName := HgF_GetTypeNameByAddress(Variable.pValue, TO_UDINT(Variable.diSize), e => e);

END_FUNCTION

// POUs/Functions/HgF_GetTypeNameByPath
// Returns the datatype of a variable as a string using its path.
FUNCTION HgF_GetTypeNameByPath : HgT_Str
VAR_INPUT
	Path : HgT_LStr; // Variable/Symbol path as string | e.g. 'MAIN.nVar'
END_VAR
VAR_OUTPUT
	e : HgT_Error;
END_VAR
VAR 
	_nTmp : UDINT := SIZEOF(HgF_GetTypeNameByPath);
	_ipComInterface : ITcIecApplicationInfo := HgF_TcComIecApplicationInfo().GetInterface(e => e);
	_Result : HRESULT;
END_VAR

IF _ipComInterface <> 0 THEN
	_Result := _ipComInterface.GetSymbolDatatype(Path, _nTmp, ADR(HgF_GetTypeNameByPath));
	e := SEL(
		Tc3_Module.SUCCEEDED(_Result),
		HgF_CreateError(TRUE, _Result, 'Failed to get variable typename. Check error code against "Tc3_Module/Error Codes" section on infosys.', 0),
		HgGVL_Errors.NO_ERROR);
	END_IF

END_FUNCTION

// POUs/MAIN
PROGRAM INTERNAL MAIN
VAR
	i : HgT_Size;
	bHasChanged, bHasChanged2 : BOOL;
	fbObj : HgFB_Object;
	Error : HgFB_Error;
	sName, sName2, sPath, sTypeName : HgT_LStr;
	sz : HgT_Size;
	Init : HgT_FirstCall;
	ch : HgFB_CycleChanged;
	dd : UDINT := TO_UDINT(DINT#-1);
	fbHasChanged : HgFB_HasChanged;
	//fbObj2 : HgFB_Object;
	//SysInfo : HgT_SysInfo;
	//Code : HgE_ErrorCodes;
END_VAR

bHasChanged := ch._;
sz := fbObj.Size;
IF fbHasChanged.Watch(dd) THEN i := i + 1; END_IF
IF Init._ THEN 
	//...
	sPath := Init.GetInstancePath();
	sTypeName := fbObj.GetTypeName();
	sName := HgF_GetVariableName(bHasChanged);
	sName2 := HgF_GetVariableNameByPath(fbObj.GetInstancePath());
	END_IF
	
bHasChanged2 := ch._;

END_PROGRAM

// POUs/Functions/HgF_GetVariableName
// Returns the name of a variable as a string.
// Variables allocated in dynamic memory are not supported.
FUNCTION HgF_GetVariableName : HgT_LStr
VAR_INPUT
	Variable : ANY;
END_VAR
VAR_OUTPUT
	e : HgT_Error;
END_VAR

HgF_GetVariableName := HgF_GetVariableNameByAddress(Variable.pValue, TO_UDINT(Variable.diSize), e => e);

END_FUNCTION

// POUs/Functions/HgF_GetVariableNameByPath
// Returns the name of a variable as a string using its path.
FUNCTION HgF_GetVariableNameByPath : HgT_LStr
VAR_INPUT
	Path : HgT_LStr; // Variable/Symbol path as string | e.g. 'MAIN.nVar'
END_VAR
VAR_OUTPUT
	e : HgT_Error;
END_VAR
VAR
	_pCursor : POINTER TO BYTE;
	_pVariableName : POINTER TO HgT_LStr;
END_VAR

IF Path = '' THEN 
	e := HgF_CreateError(TRUE, HgE_ErrorCodes.ERR_INVALID_PARAMETER, 'Path string is empty.', 0);
	RETURN; 
	END_IF

_pCursor := ADR(Path);

REPEAT
	IF (_pCursor^ = 32) OR_ELSE (_pCursor^ = 9) OR_ELSE (_pCursor^ = 10) OR_ELSE (_pCursor^ = 13) OR_ELSE (_pCursor^ = 12) OR_ELSE (_pCursor^ = 11) THEN
		e := HgF_CreateError(TRUE, HgE_ErrorCodes.ERR_INVALID_PARAMETER, 'Path string cannot contain a space.', 0);
		RETURN;
		END_IF
	IF _pCursor^ = 46 THEN _pVariableName := _pCursor + 1; END_IF
	_pCursor := _pCursor + 1;
UNTIL
	_pCursor^ = 0
	END_REPEAT

HgF_GetVariableNameByPath := SEL(_pVariableName = 0, _pVariableName^, Path);

END_FUNCTION

// POUs/Functions/HgF_GetVariablePath
// Returns the path of a variable as a string.
// Variables allocated in dynamic memory are not supported.
FUNCTION HgF_GetVariablePath : HgT_LStr
VAR_INPUT
	Variable : ANY;
END_VAR
VAR_OUTPUT
	e : HgT_Error;
END_VAR

HgF_GetVariablePath := HgF_GetVariablePathByAddress(Variable.pValue, TO_UDINT(Variable.diSize), e => e);

END_FUNCTION

// POUs/Functions/HgF_IsAllTrue
// Checks if every boolean in array is TRUE
FUNCTION HgF_IsAllTrue : BOOL
VAR_IN_OUT
	arbItems : ARRAY[*] OF BOOL;
END_VAR
VAR
	i : DINT;
END_VAR

FOR i := LOWER_BOUND(arbItems, 1) TO UPPER_BOUND(arbItems, 1) DO
	IF arbItems[i] = FALSE THEN RETURN; END_IF 
	END_FOR
	
HgF_IsAllTrue := TRUE;

END_FUNCTION

// POUs/Functions/HgF_IsAnyTrue
// Checks if one of the boolean values in array is TRUE
FUNCTION HgF_IsAnyTrue : BOOL
VAR_IN_OUT
	arbItems : ARRAY[*] OF BOOL;
END_VAR
VAR
	i : DINT;
END_VAR

FOR i := LOWER_BOUND(arbItems, 1) TO UPPER_BOUND(arbItems, 1) DO
	IF arbItems[i] = TRUE THEN HgF_IsAnyTrue := TRUE; RETURN; END_IF 
	END_FOR

END_FUNCTION

// POUs/Functions/HgF_IsInRange
// Checks if a value is in range. Returns TRUE if it is.
FUNCTION HgF_IsInRange : BOOL
VAR_INPUT
	fLowerLimit,
	fUpperLimit,
	fValue : LREAL;
END_VAR

HgF_IsInRange := fValue >= fLowerLimit AND fValue <= fUpperLimit;

END_FUNCTION

// POUs/Functions/HgF_IsOutOfRange
// Checks if a value is out of range. Returns TRUE if it is.
FUNCTION HgF_IsOutOfRange : BOOL
VAR_INPUT
	fLowerLimit,
	fUpperLimit,
	fValue : LREAL;
END_VAR

HgF_IsOutOfRange := fValue < fLowerLimit OR fValue > fUpperLimit;

END_FUNCTION

// POUs/Functions/HgF_Lerp
// Linear interpolation (Lerp) - this function interpolates values between 2 time points in 1D space.
// The equation is Lerp(Point A, Point B, Percentage) = Point A + (Point B - Point A) * Percentage.
// Any value between the 2 points can be represented through a percentage.
FUNCTION HgF_Lerp : LREAL
VAR_INPUT
	fA : LREAL; // Point A.
	fB : LREAL; // Point B.
	fPercentage : LREAL; // 0.14 = 14%.
END_VAR

HgF_Lerp := fA + (fB - fA) * fPercentage;

END_FUNCTION

// POUs/Functions/HgF_ResetFlagIfTrue
// Sets the input to false if true. 
// Returns true if input was true, otherwise false.
FUNCTION HgF_ResetFlagIfTrue : BOOL
VAR_INPUT
	bInput : REFERENCE TO BOOL;
END_VAR

IF bInput THEN bInput := FALSE; HgF_ResetFlagIfTrue := TRUE;END_IF

END_FUNCTION

// POUs/Programs/HgP_SystemInformation
{attribute 'no_explicit_call' := 'direct call for this program is not allowed'} 
PROGRAM HgP_SystemInformation

// The version as defined in the compile options.
PROPERTY CompilerVersion : VERSION
GET
CompilerVersion := __SYSTEM.Constants.CompilerVersion;
END_GET
END_PROPERTY

// The version as defined in the compile options.
PROPERTY CompilerVersionNumeric : DWORD
GET
CompilerVersionNumeric := __SYSTEM.Constants.CompilerVersionNumeric;
END_GET
END_PROPERTY

// Indication of whether the target has FPU support | Supported = TRUE.
PROPERTY HasFpuSupport : BOOL
GET
HasFpuSupport := __SYSTEM.Constants.bFPUSupport;
END_GET
END_PROPERTY

// Indicates whether multicore support is available in the target | Multicore supported = TRUE.
PROPERTY HasMulticoreSupport : BOOL
GET
HasMulticoreSupport := __SYSTEM.Constants.bMulticoreSupport;
END_GET
END_PROPERTY

// Indicates if system is in simulation mode | Simulation mode = TRUE.
PROPERTY InSimulationMode : BOOL
GET
InSimulationMode := __SYSTEM.Constants.bSimulationMode;
END_GET
END_PROPERTY

// Indicates of the system is little endian | TRUE for Intel, ARM etc. FALSE for PPC etc. 
PROPERTY IsLittleEndian : BOOL
GET
IsLittleEndian := __SYSTEM.Constants.bLittleEndian;
END_GET
END_PROPERTY

// Retrieves the packmode of the system.
PROPERTY PackMode : WORD
GET
PackMode := __SYSTEM.Constants.nPackMode;
END_GET
END_PROPERTY

// Retrieves the size of the CPU register | 16 for C16x, 64 for X86-64 Bit, 32 for all other controllers.
PROPERTY RegisterSize : WORD
GET
RegisterSize := __SYSTEM.Constants.nRegisterSize;
END_GET
END_PROPERTY

// The version as described in the runtime system.
PROPERTY RuntimeVersion : VERSION
GET
RuntimeVersion := __SYSTEM.Constants.RuntimeVersion;
END_GET
END_PROPERTY

// The version as described in the runtime system.
PROPERTY RuntimeVersionNumeric : DWORD
GET
RuntimeVersionNumeric := __SYSTEM.Constants.RuntimeVersionNumeric;
END_GET
END_PROPERTY

END_PROGRAM

// Project Information/F_GetCompany
// This function has been automatically generated from the project information.
{attribute 'signature_flag' := '1073741824'}
{attribute 'TcGenerated'}
{attribute 'no-analysis'}
FUNCTION F_GetCompany : WSTRING
VAR_INPUT
	
END_VAR

F_GetCompany := "Johnson Matthey Technology Centre";

END_FUNCTION

// Project Information/F_GetTitle
// This function has been automatically generated from the project information.
{attribute 'signature_flag' := '1073741824'}
{attribute 'TcGenerated'}
{attribute 'no-analysis'}
FUNCTION F_GetTitle : WSTRING
VAR_INPUT
	
END_VAR

F_GetTitle := "Hg_Core";

END_FUNCTION

// Project Information/F_GetVersion
// This function has been automatically generated from the project information.
{attribute 'signature_flag' := '1073741824'}
{attribute 'TcGenerated'}
{attribute 'no-analysis'}
FUNCTION F_GetVersion : ST_LibVersion
VAR_INPUT
	
END_VAR

F_GetVersion.iMajor := 0;
F_GetVersion.iMinor := 0;
F_GetVersion.iBuild := 0;
F_GetVersion.iRevision := 17;

END_FUNCTION
